(* CODESYS project interlock.project

Project tree, tasks and I/O mapping:
  Device : AC702, Shenzhen Inovance Technology Co., Ltd., version 3.5.11.51
    application Application
      libraries: Standard, * (System)
      task MainTask (cyclic, interval 20 ms, priority 2) calls PLC_PRG
      trace Trace (task ): PLC_PRG.motorF
      DifferentialMonitor
      program PLC_PRG [LD]
    HardWare Configuration
    Network Configuration
    Device Diagnosis
    Resources List
    ConfigStorage
    SoftMotion General Axis Pool
    LocalHSIO : 本地高速IO, 汇川技术股份有限公司, version 1.0.0.0
        unmapped channels: DigitalInput, DigitalOutput
    MODBUS_TCP : ModbusTCP本地从站, inovance, version 00.00.00.10
    HwConfiguratioinDevice : SystemConfig, Inovance, version 00.00.00.10
        settings: NetworkConfigArray.NetworkConfigArray.BusType = 10; NetworkConfigArray.NetworkConfigArray.RackSum = 1; NetworkConfigArray.NetworkConfigArray.HardwareConfigArray.HardwareConfigArray.RackNo = 1
*)

// Device/Application/PLC_PRG
PROGRAM PLC_PRG
VAR
	fwd: BOOL;
	rev: BOOL;
	stop: BOOL;
	motorF: BOOL;
	motorR: BOOL;
END_VAR

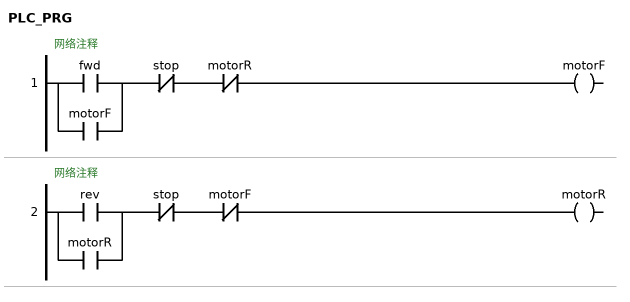
// NETWORK 1
// 网络注释
motorF := (fwd OR motorF) AND NOT stop AND NOT motorR;

// NETWORK 2
// 网络注释
motorR := (rev OR motorR) AND NOT stop AND NOT motorF;

END_PROGRAM
